(* IEC 61131-3 sources: Industry-PLC-LLM/data/PLCBEAD_repo/PLCBEAD_PLCEmbed-main/PLC-BEAD/Source/GEB/TEMP_NI, 1 file *)

(* ---- TEMP_NI.ST ---- *)
FUNCTION TEMP_NI:REAL
	VAR_INPUT
		RES :	REAL;
		R0 :	REAL;
	END_VAR

	TEMP_NI := (SQRT(0.30085225 - 2.66E-3 * (R0 - Res)) - 0.5485) * 751.8796992;
END_FUNCTION

PROGRAM program0
  	VAR
		RES :	REAL;
		R0 :	REAL;
    	CEIL5_OUT : REAL;
  	END_VAR

  	CEIL5_OUT := TEMP_NI(RES, R0);
END_PROGRAM
